# EPICS substitutions: ek9000App/Db/EL4022.substitutions
file EL4022.template
{       pattern
        {
                TERMINAL,

        }
        {
        }
}
